(* Schneider Machine Expert - Basic project resolucao, file version 2.7.0.0 *)
(* ProjectInformations: Name=Novo projeto *)

HARDWARE
  Cpu 0: TM221C24R
  EthernetConfiguration: NetworkName=M221, IpAllocationMode=FixedAddress, IpAddress=0.0.0.0, SubnetMask=0.0.0.0
  SerialLineConfiguration: Baud=Baud19200, Parity=ParityEven, DataBits=DataBits8, StopBits=StopBits1, PhysicalMedium=PhysicalMediumRs485, TransmissionMode=TransmissionModeModbusRtu, SlaveId=1, Addressing=SlaveAddressing
  MastTask: UsePeriodScanMode=false, PeriodScan=100
  FastTask: Period=255
  CpuBehavior: StartingMode=StartAsPreviousState, AutoSaveRamOnEeprom=true, WatchdogPeriod=250

SYMBOLS  (address, symbol, comment, settings)
  %M0       SIG_E1_E2
  %M1       SIG_E2_E3
  %M2       SIG_E3_E4
  %M3       SIG_E4_E1
  %M11      SIG_OUT_SEM_HOR_VERD
  %M12      SIG_OUT_SEM_HOR_AMA
  %M13      SIG_OUT_SEM_HOR_VERM
  %M15      SIG_OUT_SEM_VERT_VERD
  %M16      SIG_OUT_SEM_VERT_AMA
  %M17      SIG_OUT_SEM_VERT_VERM
  %TM0      FT_E1_E2  [Preset=10, Base=OneSecond]
  %TM1      FT_E2_E3  [Preset=3, Base=OneSecond]
  %TM2      FT_E3_E4  [Preset=10, Base=OneSecond]
  %TM3      FT_E4_E1  [Preset=3, Base=OneSecond]
  %Q0.1     OUT_SEM_HOR_VERD
  %Q0.2     OUT_SEM_HOR_AMA
  %Q0.3     OUT_SEM_HOR_VERM
  %Q0.5     OUT_SEM_VERT_VERD
  %Q0.6     OUT_SEM_VERT_AMA
  %Q0.7     OUT_SEM_VERT_VERM

GRAFCET Grafcet POU
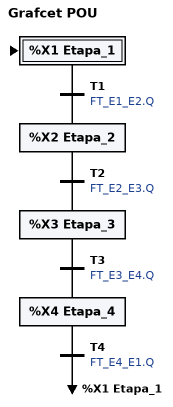
  INITIAL_STEP %X1  (* Etapa_1 *)
  STEP %X2  (* Etapa_2 *)
  STEP %X3  (* Etapa_3 *)
  STEP %X4  (* Etapa_4 *)
  TRANSITION T1 FROM %X1 TO %X2 := FT_E1_E2.Q;
  TRANSITION T2 FROM %X2 TO %X3 := FT_E2_E3.Q;
  TRANSITION T3 FROM %X3 TO %X4 := FT_E3_E4.Q;
  TRANSITION T4 FROM %X4 TO %X1 := FT_E4_E1.Q;

STEP %X1 Etapa_1
  (* SectionNumber=1, StepNumber=1 *)

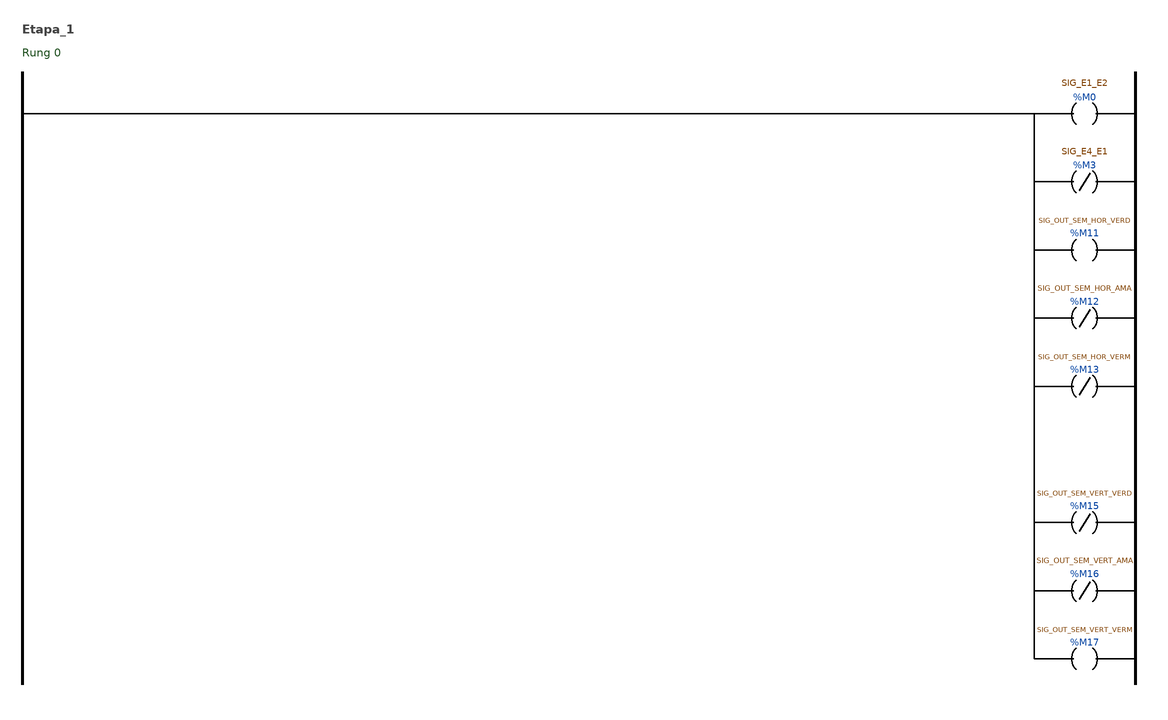

// Rung 0
  LD 1
  ST %M0                  (* SIG_E1_E2 *)
  STN %M3                 (* SIG_E4_E1 *)
  ST %M11                 (* SIG_OUT_SEM_HOR_VERD *)
  STN %M12                (* SIG_OUT_SEM_HOR_AMA *)
  STN %M13                (* SIG_OUT_SEM_HOR_VERM *)
  STN %M15                (* SIG_OUT_SEM_VERT_VERD *)
  STN %M16                (* SIG_OUT_SEM_VERT_AMA *)
  ST %M17                 (* SIG_OUT_SEM_VERT_VERM *)
  // as ST:
  //   SIG_E1_E2 := TRUE;
  //   SIG_E4_E1 := FALSE;
  //   SIG_OUT_SEM_HOR_VERD := TRUE;
  //   SIG_OUT_SEM_HOR_AMA := FALSE;
  //   SIG_OUT_SEM_HOR_VERM := FALSE;
  //   SIG_OUT_SEM_VERT_VERD := FALSE;
  //   SIG_OUT_SEM_VERT_AMA := FALSE;
  //   SIG_OUT_SEM_VERT_VERM := TRUE;

STEP %X2 Etapa_2
  (* SectionNumber=2, StepNumber=2 *)

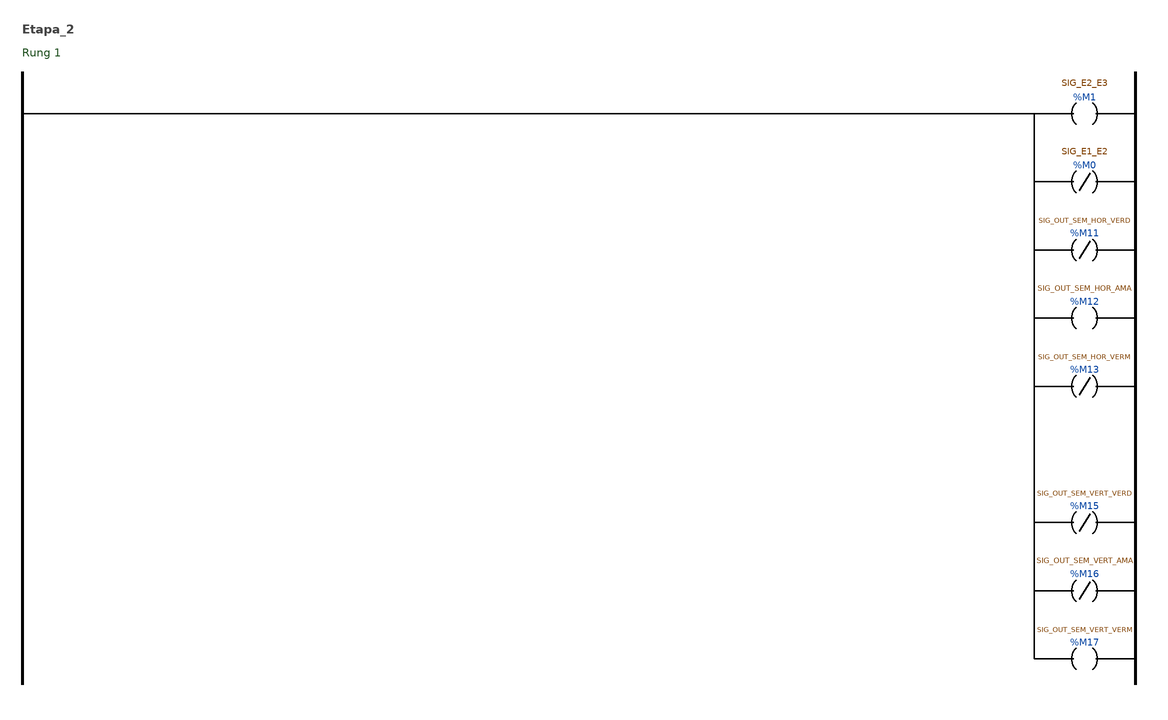

// Rung 1
  LD 1
  ST %M1                  (* SIG_E2_E3 *)
  STN %M0                 (* SIG_E1_E2 *)
  STN %M11                (* SIG_OUT_SEM_HOR_VERD *)
  ST %M12                 (* SIG_OUT_SEM_HOR_AMA *)
  STN %M13                (* SIG_OUT_SEM_HOR_VERM *)
  STN %M15                (* SIG_OUT_SEM_VERT_VERD *)
  STN %M16                (* SIG_OUT_SEM_VERT_AMA *)
  ST %M17                 (* SIG_OUT_SEM_VERT_VERM *)
  // as ST:
  //   SIG_E2_E3 := TRUE;
  //   SIG_E1_E2 := FALSE;
  //   SIG_OUT_SEM_HOR_VERD := FALSE;
  //   SIG_OUT_SEM_HOR_AMA := TRUE;
  //   SIG_OUT_SEM_HOR_VERM := FALSE;
  //   SIG_OUT_SEM_VERT_VERD := FALSE;
  //   SIG_OUT_SEM_VERT_AMA := FALSE;
  //   SIG_OUT_SEM_VERT_VERM := TRUE;

TRANSITION T1 (%X1 -> %X2) 
  (* SectionNumber=0 *)

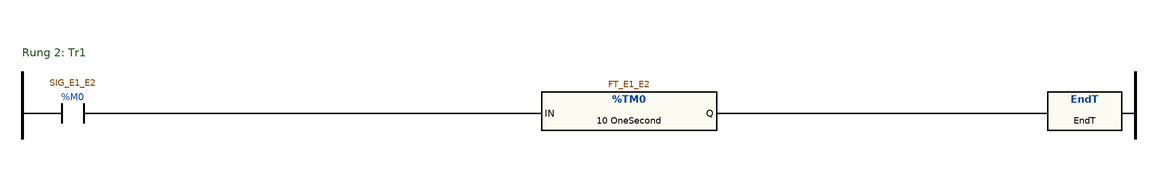

// Rung 2: Tr1
  BLK %TM0                (* FT_E1_E2 *)
  LD %M0                  (* SIG_E1_E2 *)
  IN
  OUT_BLK
  LD Q
  ENDT
  END_BLK
  // as ST:
  //   FT_E1_E2(IN := SIG_E1_E2);
  //   TRANSITION := FT_E1_E2.Q;

STEP %X3 Etapa_3
  (* SectionNumber=3, StepNumber=3 *)

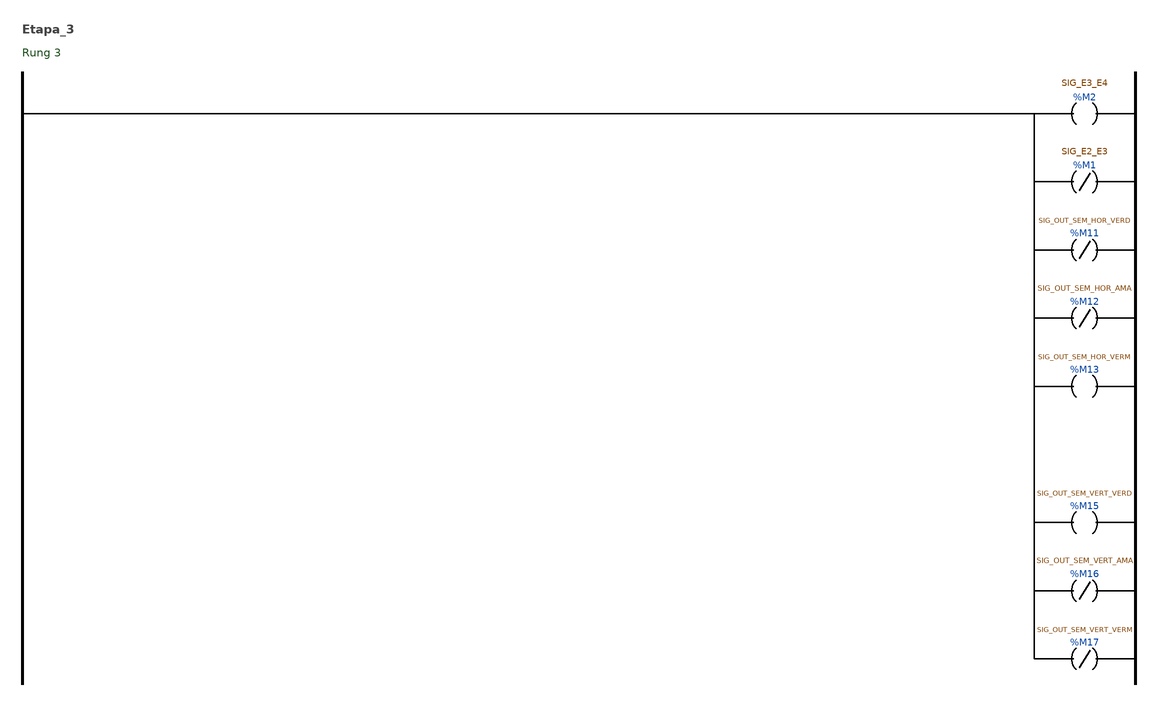

// Rung 3
  LD 1
  ST %M2                  (* SIG_E3_E4 *)
  STN %M1                 (* SIG_E2_E3 *)
  STN %M11                (* SIG_OUT_SEM_HOR_VERD *)
  STN %M12                (* SIG_OUT_SEM_HOR_AMA *)
  ST %M13                 (* SIG_OUT_SEM_HOR_VERM *)
  ST %M15                 (* SIG_OUT_SEM_VERT_VERD *)
  STN %M16                (* SIG_OUT_SEM_VERT_AMA *)
  STN %M17                (* SIG_OUT_SEM_VERT_VERM *)
  // as ST:
  //   SIG_E3_E4 := TRUE;
  //   SIG_E2_E3 := FALSE;
  //   SIG_OUT_SEM_HOR_VERD := FALSE;
  //   SIG_OUT_SEM_HOR_AMA := FALSE;
  //   SIG_OUT_SEM_HOR_VERM := TRUE;
  //   SIG_OUT_SEM_VERT_VERD := TRUE;
  //   SIG_OUT_SEM_VERT_AMA := FALSE;
  //   SIG_OUT_SEM_VERT_VERM := FALSE;

TRANSITION T2 (%X2 -> %X3) 
  (* SectionNumber=0 *)

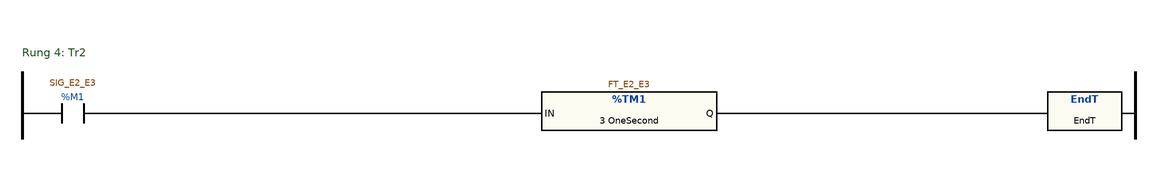

// Rung 4: Tr2
  BLK %TM1                (* FT_E2_E3 *)
  LD %M1                  (* SIG_E2_E3 *)
  IN
  OUT_BLK
  LD Q
  ENDT
  END_BLK
  // as ST:
  //   FT_E2_E3(IN := SIG_E2_E3);
  //   TRANSITION := FT_E2_E3.Q;

STEP %X4 Etapa_4
  (* SectionNumber=4, StepNumber=4 *)

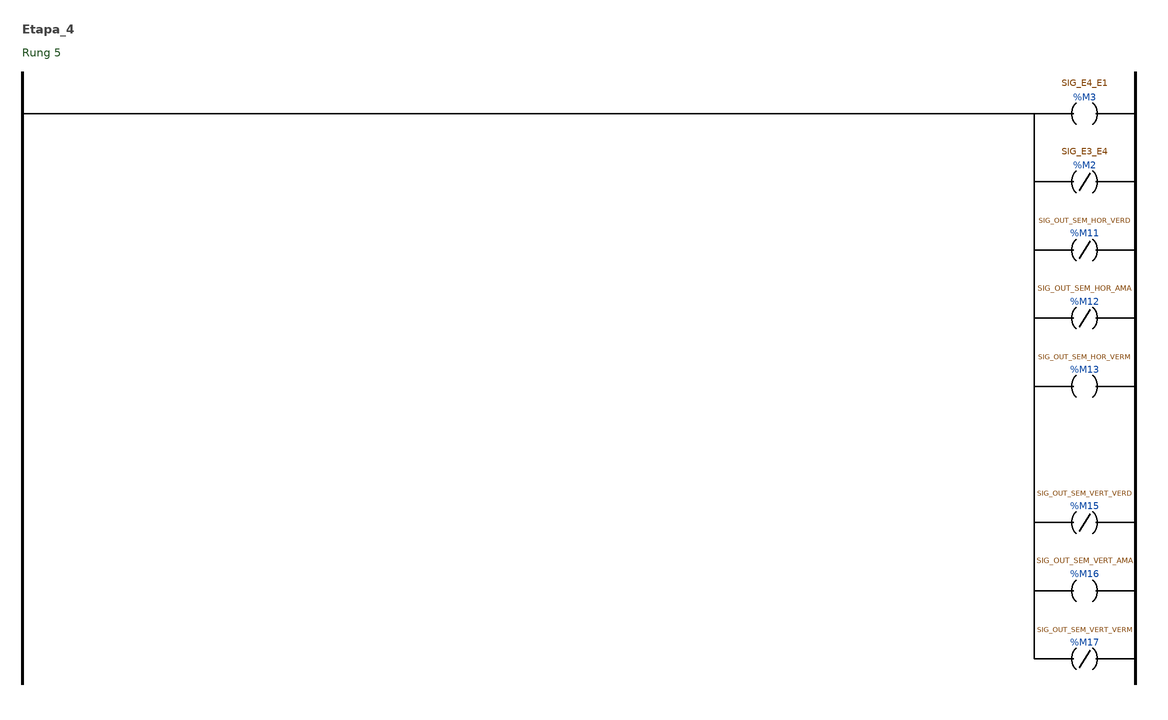

// Rung 5
  LD 1
  ST %M3                  (* SIG_E4_E1 *)
  STN %M2                 (* SIG_E3_E4 *)
  STN %M11                (* SIG_OUT_SEM_HOR_VERD *)
  STN %M12                (* SIG_OUT_SEM_HOR_AMA *)
  ST %M13                 (* SIG_OUT_SEM_HOR_VERM *)
  STN %M15                (* SIG_OUT_SEM_VERT_VERD *)
  ST %M16                 (* SIG_OUT_SEM_VERT_AMA *)
  STN %M17                (* SIG_OUT_SEM_VERT_VERM *)
  // as ST:
  //   SIG_E4_E1 := TRUE;
  //   SIG_E3_E4 := FALSE;
  //   SIG_OUT_SEM_HOR_VERD := FALSE;
  //   SIG_OUT_SEM_HOR_AMA := FALSE;
  //   SIG_OUT_SEM_HOR_VERM := TRUE;
  //   SIG_OUT_SEM_VERT_VERD := FALSE;
  //   SIG_OUT_SEM_VERT_AMA := TRUE;
  //   SIG_OUT_SEM_VERT_VERM := FALSE;

TRANSITION T3 (%X3 -> %X4) 
  (* SectionNumber=0 *)

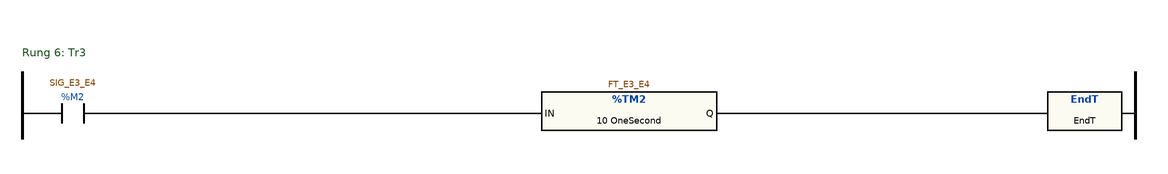

// Rung 6: Tr3
  BLK %TM2                (* FT_E3_E4 *)
  LD %M2                  (* SIG_E3_E4 *)
  IN
  OUT_BLK
  LD Q
  ENDT
  END_BLK
  // as ST:
  //   FT_E3_E4(IN := SIG_E3_E4);
  //   TRANSITION := FT_E3_E4.Q;

TRANSITION T4 (%X4 -> %X1) 
  (* SectionNumber=0 *)

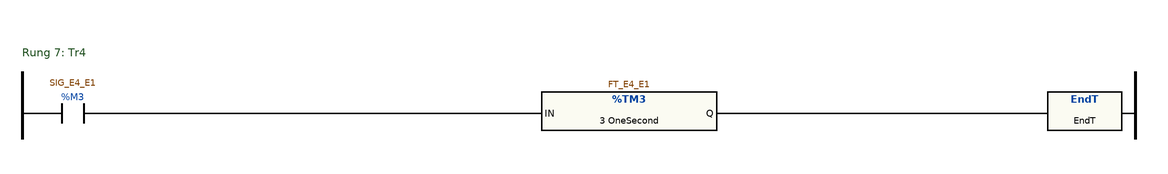

// Rung 7: Tr4
  BLK %TM3                (* FT_E4_E1 *)
  LD %M3                  (* SIG_E4_E1 *)
  IN
  OUT_BLK
  LD Q
  ENDT
  END_BLK
  // as ST:
  //   FT_E4_E1(IN := SIG_E4_E1);
  //   TRANSITION := FT_E4_E1.Q;

POU Saídas
  (* SectionNumber=6 *)

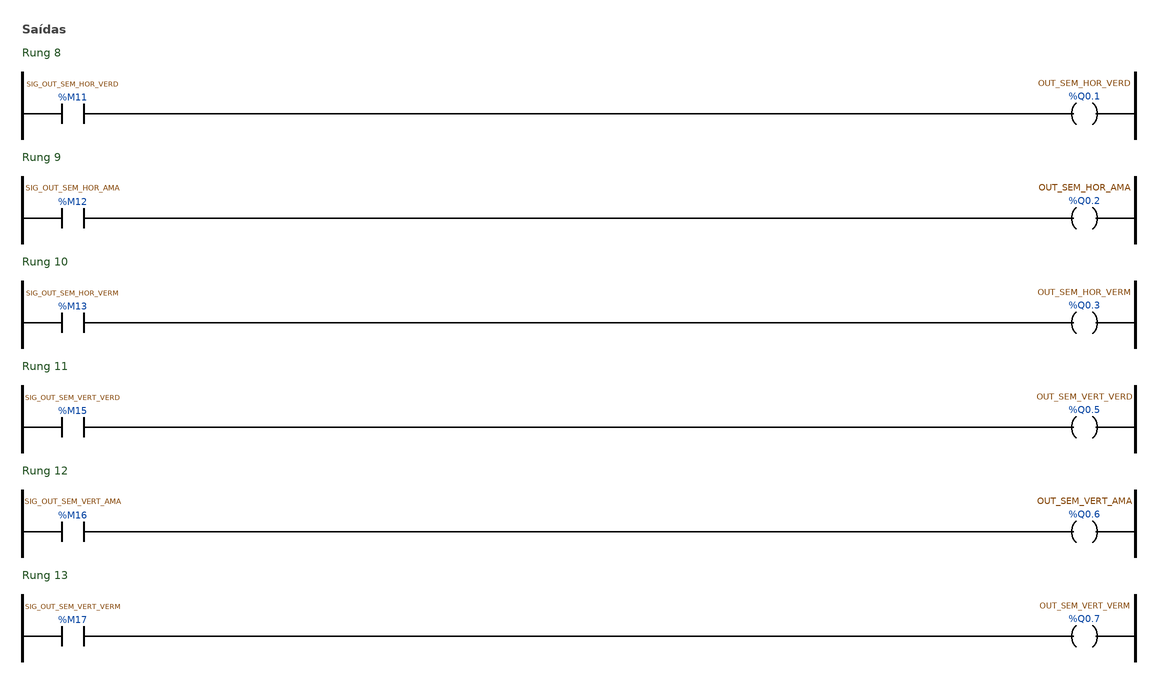

// Rung 8
  LD %M11                 (* SIG_OUT_SEM_HOR_VERD *)
  ST %Q0.1                (* OUT_SEM_HOR_VERD *)
  // as ST:
  //   OUT_SEM_HOR_VERD := SIG_OUT_SEM_HOR_VERD;

// Rung 9
  LD %M12                 (* SIG_OUT_SEM_HOR_AMA *)
  ST %Q0.2                (* OUT_SEM_HOR_AMA *)
  // as ST:
  //   OUT_SEM_HOR_AMA := SIG_OUT_SEM_HOR_AMA;

// Rung 10
  LD %M13                 (* SIG_OUT_SEM_HOR_VERM *)
  ST %Q0.3                (* OUT_SEM_HOR_VERM *)
  // as ST:
  //   OUT_SEM_HOR_VERM := SIG_OUT_SEM_HOR_VERM;

// Rung 11
  LD %M15                 (* SIG_OUT_SEM_VERT_VERD *)
  ST %Q0.5                (* OUT_SEM_VERT_VERD *)
  // as ST:
  //   OUT_SEM_VERT_VERD := SIG_OUT_SEM_VERT_VERD;

// Rung 12
  LD %M16                 (* SIG_OUT_SEM_VERT_AMA *)
  ST %Q0.6                (* OUT_SEM_VERT_AMA *)
  // as ST:
  //   OUT_SEM_VERT_AMA := SIG_OUT_SEM_VERT_AMA;

// Rung 13
  LD %M17                 (* SIG_OUT_SEM_VERT_VERM *)
  ST %Q0.7                (* OUT_SEM_VERT_VERM *)
  // as ST:
  //   OUT_SEM_VERT_VERM := SIG_OUT_SEM_VERT_VERM;
